// TIA Portal V21 export
TYPE "coneCrusherAlm"
   STRUCT
      stepErr : Bool;
      extStop : Bool;
      emStop : Bool;
      premolding : Bool;
      sgFault : Bool;
      luSNotRun : Bool;
      preStAlmNoFb : Bool;
      preStAlmFalseFb : Bool;
      returnOilTempHiHi : Bool;
      noKeySwitch : Bool;
      crusherEccentricTempHiHi : Bool;
      crusherOuterBearingTempHiHi { S7_SetPoint := 'True'} : Bool;
      crusherInnerBearingTempHiHi { S7_SetPoint := 'True'} : Bool;
      driveFrontBearingTempHiHi { S7_SetPoint := 'True'} : Bool;
      driveRearBearingTempHiHi { S7_SetPoint := 'True'} : Bool;
      driveWindingTempP1HiHi { S7_SetPoint := 'True'} : Bool;
      driveWindingTempP2HiHi { S7_SetPoint := 'True'} : Bool;
      driveWindingTempP3HiHi { S7_SetPoint := 'True'} : Bool;
      driveCurrentHiHi { S7_SetPoint := 'True'} : Bool;
   END_STRUCT;
END_TYPE
